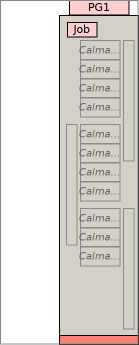
VISUALIZATION _VISU_PmEnable_Maxliner  // 139x345
VAR_IN_OUT
  mInst : FB_PrintModule_Maxliner;
END_VAR
    RoundedRectangle (59,15 80x329), tooltip "WorkerPrint enable"
        toggle mInst.fbWorkerPrint[1]._bEnable
    RoundedRectangle (69,0 60x15), "PG1", tooltip "PG enable"
        toggle mInst.fbWorkerPrint[1]._pAdsPg^.stAds.bI_Enable
    Frame (123,40 11x121)
        shows CalmarCompPrint._VISU_PC_MiniVertical(mInst := mInst._pPc[1]^)
    Frame (66,124 11x121)
        shows CalmarCompPrint._VISU_PC_MiniVertical(mInst := mInst._pPc[2]^)
    Frame (80,40 40x20)
        shows CalmarCompPrint._VISU_PH_TinyVertical(mInst := mInst._pPh[1]^)
    Frame (80,59 40x20)
        shows CalmarCompPrint._VISU_PH_TinyVertical(mInst := mInst._pPh[2]^)
    Frame (80,78 40x20)
        shows CalmarCompPrint._VISU_PH_TinyVertical(mInst := mInst._pPh[3]^)
    Frame (80,97 40x20)
        shows CalmarCompPrint._VISU_PH_TinyVertical(mInst := mInst._pPh[4]^)
    Frame (80,124 40x20)
        shows CalmarCompPrint._VISU_PH_TinyVertical(mInst := mInst._pPh[5]^)
    Frame (80,143 40x20)
        shows CalmarCompPrint._VISU_PH_TinyVertical(mInst := mInst._pPh[6]^)
    RoundedRectangle (67,22 30x15), "Job", tooltip "Job is active", colour toggle: mInst.fbWorkerPrint[1]._bJobActive
    RoundedRectangle (59,335 80x10), tooltip "Worker PrintEnable"
        toggle mInst.fbWorkerPrint[1].bWorkerPrintEnable
    Frame (80,162 40x20)
        shows CalmarCompPrint._VISU_PH_TinyVertical(mInst := mInst._pPh[7]^)
    Frame (80,181 40x20)
        shows CalmarCompPrint._VISU_PH_TinyVertical(mInst := mInst._pPh[8]^)
    Frame (123,208 11x121)
        shows CalmarCompPrint._VISU_PC_MiniVertical(mInst := mInst._pPc[3]^)
    Frame (80,208 40x20)
        shows CalmarCompPrint._VISU_PH_TinyVertical(mInst := mInst._pPh[9]^)
    Frame (80,227 40x20)
        shows CalmarCompPrint._VISU_PH_TinyVertical(mInst := mInst._pPh[10]^)
    Frame (80,246 40x20)
        shows CalmarCompPrint._VISU_PH_TinyVertical(mInst := mInst._pPh[11]^)
END_VISUALIZATION

(* stored: Version 1.1.0.1, ProductVersion 3.1.4024.11
   Visu _VISU_PmEnable_Maxliner: Id {cecfd759-7f37-44c5-a301-18f2086cfe0e} *)
